// TwinCAT 3 PLC project TcLog_Test
// ProgramVersion: 3.1.4026.20
// libraries:
//   Tc2_Standard, * (Beckhoff Automation GmbH)
//   Tc2_System, * (Beckhoff Automation GmbH)
//   Tc2_Utilities, * (Beckhoff Automation GmbH)
//   Tc3_Module, * (Beckhoff Automation GmbH)
//   [TcLog], * (Benedikt Geisler)
//   TcUnit, * (www.tcunit.org)
// project tree:
//   Tasks/ PlcTask.TcTTO
//   TestRunners/ TestRunner.TcPOU, TestWrapper.TcPOU
//   Tests/ ConvertAnyToString_Test.TcPOU, DateTime_Test.TcPOU, DynamicStringBuffer_Test.TcPOU
// real-time tasks:
//   TASK PlcTask1: cycle T#10ms, priority 21, ADS port 351

CONFIGURATION TcLog_Test
    RESOURCE PLC ON TwinCAT3
        TASK PlcTask(INTERVAL := T#10ms, PRIORITY := 21);
        PROGRAM TestRunner WITH PlcTask : TestRunner;
    END_RESOURCE
END_CONFIGURATION

// ---- TestRunners/TestRunner.TcPOU
PROGRAM TestRunner
VAR
	test_wrapper : TestWrapper;
	date_time_time : DateTime_Test;
	helper_functions_test : ConvertAnyToString_Test;
	dynamic_string_buffer_test : DynamicStringBuffer_Test;
END_VAR

test_wrapper();

TcUnit.Run();

END_PROGRAM

// ---- TestRunners/TestWrapper.TcPOU
FUNCTION_BLOCK TestWrapper
VAR
	core_logger : TcLogCore(BufferSize:=50 * 50 * (Tc2_System.MAX_STRING_LENGTH + Constants.FifoOverhead));
	core_logger_first_cycle : TcLogCore(BufferSize:=50 * 50 * (Tc2_System.MAX_STRING_LENGTH + Constants.FifoOverhead));
	core_logger_first_cycle_valid_timestamp_only : TcLogCore(BufferSize:=50 * 50 * (Tc2_System.MAX_STRING_LENGTH + Constants.FifoOverhead));
	logger_first_cycle : TcLog;
	logger_first_cycle_valid_timestamp_only : TcLog;
	logger : TcLog;
	flush_cache : BOOL;
	ads_adapter : AdsLogTargetAdapter;
 
	// Test drivers
	date_time : DateTime;
	set_local_system_time : NT_SetLocalTime;
	cycles : INT;
	_i : INT;
	persistence_time_stays_within_bounds : F_Trig;
	is_first_cycle: BOOL := TRUE;
	
	// Exchanged variables with .NET tests
	FilePath : STRING;
	FileName : STRING;
	Delimiter : STRING(1);
	NewLocalSystemTimeToBeSet : STRING;
	TriggerNewLocalSystemTime : BOOL;
	LocalTimeAsString : STRING;
	
	Persist_simple_error_message_run : BOOL;
	Persist_simple_error_message_data : STRING;
	
	Persist_long_error_message_run : BOOL;
	Persist_long_error_message_data : T_MaxString;
	
	Linebreak_is_included_when_log_message_has_maximum_length_run : BOOL;
	Linebreak_is_included_when_log_message_has_maximum_length_data : T_MaxString;
	
	Do_not_persist_logs_below_log_level_run : BOOL;
	
	Log_message_contains_instance_path_run : BOOL;
	
	Log_message_uses_correct_delimiter_run : BOOL;
	Log_message_uses_correct_delimiter_data : STRING;
	
	Log_message_contains_custom_formatted_timestamp_run : BOOL;
	
	Delete_logs_if_expired_run : BOOL;
	
	New_logfile_is_created_if_rolling_interval_rolls_run : BOOL;
	
	Same_log_file_is_used_until_rolling_interval_rolls : BOOL;
	
	Log_in_consecutive_cycles : BOOL;
	Number_of_log_cycles : DINT;
	
	Log_multiple_logs_in_one_cycle : BOOL;
	Number_of_logs_per_cycle : DINT;
	
	Log_multiple_logs_in_multiple_cycles : BOOL;
	Number_of_cycles : DINT;
	CycleCount : DINT := 1;
	
	Persistance_time_stays_within_bounds : BOOL;
	Duration_in_cylces : DINT := 1;
END_VAR

// ****** U N I T   T E S T S ******

// Set up TcLog
core_logger
	.IncludeInstancePath()
	.MinimumLevel(LogLevel.Debug)
	.SetDelimiter(Delimiter)
	.SetRollingInterval(RollingIntervals.Hourly)
	.DeleteLogFilesAfterDays(1)
	.TimestampFormat('_YYMMDD-hh-mm-ss_')
	.WriteToAds()
	.WriteToFile('C:\Log Files', 'tclog_test.log')
	.WriteToAdapter(ads_adapter)
	.RunLogger();
//logger.SetLogger(core_logger);

IF flush_cache THEN
	core_logger.FlushCache();
END_IF
  
// Test drivers
date_time.CyclicCall();
LocalTimeAsString := date_time.AsLocalSystemTimeString;

set_local_system_time(
	NetId   := '',
	TimeStr := STRING_TO_SYSTEMTIME(NewLocalSystemTimeToBeSet),
	Start   := TriggerNewLocalSystemTime,
	TmOut := T#2S
);

// Execute tests
IF Persist_simple_error_message_run THEN
	Persist_simple_error_message_run := FALSE;
	logger.Error(Persist_simple_error_message_data);
END_IF

IF Persist_long_error_message_run THEN
	Persist_long_error_message_run := FALSE;
	logger.ToCustomFormat(Persist_long_error_message_data);
END_IF

IF Linebreak_is_included_when_log_message_has_maximum_length_run THEN
	Linebreak_is_included_when_log_message_has_maximum_length_run := FALSE;
	logger
		.ToCustomFormat(Linebreak_is_included_when_log_message_has_maximum_length_data);
	logger.ToCustomFormat(Linebreak_is_included_when_log_message_has_maximum_length_data);
END_IF

IF Do_not_persist_logs_below_log_level_run THEN
	Do_not_persist_logs_below_log_level_run := FALSE;
	logger.Information('Nothing');
END_IF

IF Log_message_contains_instance_path_run THEN
	Log_message_contains_instance_path_run := FALSE;
	logger.Error('Nothing');
END_IF

IF Log_message_uses_correct_delimiter_run THEN
	Log_message_uses_correct_delimiter_run := FALSE;
	logger.Error(Log_message_uses_correct_delimiter_data);
END_IF

IF Log_message_contains_custom_formatted_timestamp_run THEN
	Log_message_contains_custom_formatted_timestamp_run := FALSE;
	logger.Error('Test message');
END_IF

IF Delete_logs_if_expired_run THEN
	Delete_logs_if_expired_run := FALSE;
	logger.Error('Test message');
END_IF

IF New_logfile_is_created_if_rolling_interval_rolls_run THEN
	New_logfile_is_created_if_rolling_interval_rolls_run := FALSE;
	logger.Error('Test message');
END_IF

IF Same_log_file_is_used_until_rolling_interval_rolls THEN
	Same_log_file_is_used_until_rolling_interval_rolls := FALSE;
	logger.Error('Test message');
END_IF

IF Log_in_consecutive_cycles THEN
	logger.Error(Tc2_Standard.CONCAT('Logging cycle ', INT_TO_STRING(cycles)));
	cycles := cycles + 1;
	IF cycles >= Number_of_log_cycles THEN
		cycles := 0;
		Log_in_consecutive_cycles := FALSE;
	END_IF
END_IF

IF Log_multiple_logs_in_one_cycle THEN
	FOR _i:= 1 TO DINT_TO_INT(Number_of_logs_per_cycle) DO
		logger.
			Error(Tc2_Standard.CONCAT('Logging multiple times per cycle. Current step: ', INT_TO_STRING(_i))); 
	END_FOR
	Log_multiple_logs_in_one_cycle := FALSE;
END_IF

IF Log_multiple_logs_in_multiple_cycles THEN
	IF CycleCount <= Number_of_cycles THEN  
		FOR _i:= 1 TO DINT_TO_INT(Number_of_logs_per_cycle) DO
			logger
				.AppendString('Logging multiple times per cycle. Cycle: ')
				.AppendString(DINT_TO_STRING(CycleCount))
				.AppendString(' / Step: ')
				.AppendString(INT_TO_STRING(_i))
				.Error('');
		END_FOR
		CycleCount := CycleCount + 1;
	ELSE
		CycleCount := 1;
		Log_multiple_logs_in_multiple_cycles := FALSE;
	END_IF
END_IF 

persistence_time_stays_within_bounds(CLK := (Persistance_time_stays_within_bounds AND core_logger.Busy));
IF persistence_time_stays_within_bounds.Q THEN
	CycleCount := 1;
	Persistance_time_stays_within_bounds := FALSE;
END_IF

IF Persistance_time_stays_within_bounds THEN
	Duration_in_cylces := Duration_in_cylces + 1;
	IF CycleCount <= Number_of_cycles THEN  
		FOR _i:= 1 TO DINT_TO_INT(Number_of_logs_per_cycle) DO
			logger
				.AppendString('Logging multiple times per cycle. Cycle: ')
				.AppendString(DINT_TO_STRING(CycleCount))
				.AppendString(' / Step: ')
				.AppendString(INT_TO_STRING(_i))
				.Error('');
		END_FOR
		CycleCount := CycleCount + 1;
	END_IF
END_IF

// Check first cpu cycle
core_logger_first_cycle
	.IncludeInstancePath()
	.MinimumLevel(LogLevel.Warning)
	.SetDelimiter(Delimiter)
	.SetRollingInterval(RollingIntervals.Hourly)
	.DeleteLogFilesAfterDays(1)
	.TimestampFormat('_YYYYMMDD-hh-mm-ss_')
	.WriteToAds()
	.WriteToFile('C:\UnitTestFirstCycle\', 'firstCycle.txt')
	.RunLogger();
logger_first_cycle.SetLogger(core_logger_first_cycle);

core_logger_first_cycle_valid_timestamp_only
	.IncludeInstancePath()
	.MinimumLevel(LogLevel.Warning)
	.SetDelimiter(Delimiter)
	.SetRollingInterval(RollingIntervals.Hourly)
	.DeleteLogFilesAfterDays(1)
	.TimestampFormat('_YYYYMMDD-hh-mm-ss_')
	.WriteToAds()
	.WriteToFile('C:\UnitTestFirstCycle\', 'firstCycleValidTimestampOnly.txt')
	.ValidTimestampsOnly()
	.RunLogger();
logger_first_cycle_valid_timestamp_only.SetLogger(core_logger_first_cycle_valid_timestamp_only);

IF is_first_cycle THEN
	logger_first_cycle.Error('Log in first cycle');
	logger_first_cycle_valid_timestamp_only.Error('Log in first cycle with valid timestamps only');
	is_first_cycle := FALSE;
END_IF

END_FUNCTION_BLOCK

// ---- Tests/DateTime_Test.TcPOU
FUNCTION_BLOCK DateTime_Test EXTENDS TcUnit.FB_TestSuite

CheckStringFormat();

METHOD CheckStringFormat
VAR_INST
	date_time : DateTime;
	expected : STRING;
	result : STRING;
END_VAR
VAR
	local_system_time : Tc2_Utilities.TimeStruct;
END_VAR
date_time.CyclicCall();

Test('CheckStringFormat');

local_system_time := date_time.AsLocalSystemTime;

expected := Tc2_Standard.CONCAT('-', TO_STRING(local_system_time.wYear));
IF local_system_time.wMonth < 10 THEN
	expected := Tc2_Standard.CONCAT(expected, '0');
END_IF

expected := Tc2_Standard.CONCAT(expected, TO_STRING(local_system_time.wMonth));
IF local_system_time.wDay < 10 THEN
	expected := Tc2_Standard.CONCAT(expected, '0');
END_IF

expected := Tc2_Standard.CONCAT(expected, TO_STRING(local_system_time.wDay));
expected := Tc2_Standard.CONCAT(expected, '-');
IF local_system_time.wHour < 10 THEN
	expected := Tc2_Standard.CONCAT(expected, '0');
END_IF

expected := Tc2_Standard.CONCAT(expected, TO_STRING(local_system_time.wHour));
expected := Tc2_Standard.CONCAT(expected, ':');
IF local_system_time.wMinute < 10 THEN 
	expected := Tc2_Standard.CONCAT(expected, '0');
END_IF

expected := Tc2_Standard.CONCAT(expected, TO_STRING(local_system_time.wMinute));
expected := Tc2_Standard.CONCAT(expected, ':');
IF local_system_time.wSecond < 10 THEN
	expected := Tc2_Standard.CONCAT(expected, '0');
END_IF

expected := Tc2_Standard.CONCAT(expected, TO_STRING(local_system_time.wSecond));
expected := Tc2_Standard.CONCAT(expected, '-');
result := date_time.ToFormatString('-YYYYMMDD-hh:mm:ss-');
IF date_time.Done THEN
	AssertEquals(
		Expected  :=  expected,
		Actual    :=  result,
		Message   :=  'Time formatting failed.'
	);

  Test_Finished();
END_IF
END_METHOD

END_FUNCTION_BLOCK

// ---- Tests/ConvertAnyToString_Test.TcPOU
FUNCTION_BLOCK ConvertAnyToString_Test EXTENDS TcUnit.FB_TestSuite

ConvertAnyByteToString();
ConvertAnyDateAndTimeToString();
ConvertAnyDateToString();
ConvertAnyDIntToString();
ConvertAnyDTToString();
ConvertAnyIntToString();
ConvertAnyLIntToString();
//ConvertAnyLRealToString();
ConvertAnyLWordToString();
ConvertAnyRealToString();
ConvertAnySIntToString();
ConvertAnyStringToString();
ConvertAnyTimeToString();
ConvertAnyTODToString();
ConvertAnyUDIntToString();
ConvertAnyUIntToString();
ConvertAnyULIntToString();
ConvertAnyUSIntToString();
ConvertAnyWordToString();
ConvertAnyWStringToString();

METHOD ConvertAnyByteToString : BOOL
VAR
	inputs : ARRAY[1..4] OF BYTE := [0, 1, 128, 255];
	expectedValues : ARRAY[1..4] OF STRING := ['0', '1', '128', '255'];
	results : ARRAY[1..4] OF STRING;
	i: INT;
END_VAR
TEST('ConvertAnyByteToString');
 
FOR i := 1 TO 4 DO
  results[i] := AnyToString(inputs[i]);
  AssertEquals(Expected := expectedValues[i],
             Actual := results[i],
             Message := FormatResult(expectedValues[i], results[i])); 
END_FOR
 
TEST_FINISHED();
END_METHOD

METHOD ConvertAnyDateAndTimeToString : BOOL
VAR
	input : DATE_AND_TIME := DT#1970-01-01-00:00;
	result : STRING;
	expected : STRING := 'DT#1970-01-01-00:00:00';
END_VAR
TEST('ConvertAnyDateAndTimeToString');
 
result := AnyToString(input);
 
AssertEquals(Expected := expected,
             Actual := result,
             Message := FormatResult(expected, result));
 
TEST_FINISHED();
END_METHOD

METHOD ConvertAnyDateToString : BOOL
VAR
	input : DATE := D#1970-01-01;
	result : STRING;
	expected : STRING := 'D#1970-01-01';
END_VAR
TEST('ConvertAnyDateToString');
 
result := AnyToString(input);
 
AssertEquals(Expected := expected,
             Actual := result,
             Message := FormatResult(expected, result));
 
TEST_FINISHED();
END_METHOD

METHOD ConvertAnyDIntToString : BOOL
VAR
	inputs : ARRAY[1..7] OF DINT := [-2147483648, -1073741824, -1, 0, 1, 1073741824, 2147483647];
	expectedValues : ARRAY[1..7] OF STRING := ['-2147483648', '-1073741824', '-1', '0', '1', '1073741824', '2147483647'];
	results : ARRAY[1..7] OF STRING;
	i: INT;
END_VAR
TEST('ConvertAnyDINTToString');
 
FOR i := 1 TO 7 DO
  results[i] := AnyToString(inputs[i]);
  AssertEquals(Expected := expectedValues[i],
             Actual := results[i],
             Message := FormatResult(expectedValues[i], results[i])); 
END_FOR

TEST_FINISHED();
END_METHOD

METHOD ConvertAnyDTToString : BOOL
VAR
	input : DT := DT#1970-01-01-00:00;
	result : STRING;
	expected : STRING := 'DT#1970-01-01-00:00:00';
END_VAR
TEST('ConvertAnyDateTimeToString');
 
result := AnyToString(input);
 
AssertEquals(Expected := expected,
             Actual := result,
             Message := FormatResult(expected, result));
 
TEST_FINISHED();
END_METHOD

METHOD ConvertAnyDWordToString : BOOL
VAR
	inputs : ARRAY[1..4] OF DWORD := [0, 1, 2147483647, 4294967295];
	expectedValues : ARRAY[1..4] OF STRING := ['0', '1', '2147483647', '4294967295'];
	results : ARRAY[1..4] OF STRING;
	i: INT;
END_VAR
TEST('ConvertAnyDWordToString');
 
FOR i := 1 TO 4 DO
  results[i] := AnyToString(inputs[i]);
  AssertEquals(Expected := expectedValues[i],
             Actual := results[i],
             Message := FormatResult(expectedValues[i], results[i])); 
END_FOR
 
TEST_FINISHED();
END_METHOD

METHOD ConvertAnyIntToString : BOOL
VAR
	inputs : ARRAY[1..7] OF INT := [-32768, -18000, -1, 0, 1, 18000, 32767];
	expectedValues : ARRAY[1..7] OF STRING := ['-32768', '-18000', '-1', '0', '1', '18000', '32767'];
	results : ARRAY[1..7] OF STRING;
	i: INT;
END_VAR
TEST('ConvertAnyINTToString');

FOR i := 1 TO 7 DO
  results[i] := AnyToString(inputs[i]);
  AssertEquals(Expected := expectedValues[i],
             Actual := results[i],
             Message := FormatResult(expectedValues[i], results[i])); 
END_FOR
      
TEST_FINISHED();
END_METHOD

METHOD ConvertAnyLIntToString : BOOL
VAR
	inputs : ARRAY[1..7] OF LINT := [-2147483648, -18000, -1, 0, 1, 18000, 2147483648];
	expectedValues : ARRAY[1..7] OF STRING := ['-2147483648', '-18000', '-1', '0', '1', '18000', '2147483648'];
	results : ARRAY[1..7] OF STRING;
	i: INT;
END_VAR
TEST('ConvertAnyLINTToString');
 
FOR i := 1 TO 7 DO
  results[i] := AnyToString(inputs[i]);
  AssertEquals(Expected := expectedValues[i],
             Actual := results[i],
             Message := FormatResult(expectedValues[i], results[i])); 
END_FOR
 
TEST_FINISHED();
END_METHOD

METHOD ConvertAnyLRealToString : BOOL
VAR
	inputs : ARRAY[1..5] OF LREAL := [-1.7976931348623157E+308, -4.94065645841247E-324, 0, 4.94065645841247E-324, 1.7976931348623157E+308];
	expectedValues : ARRAY[1..5] OF STRING := ['-1.7976931348623157E308', '-4.94065645841247E324', '0.0', '4.94065645841247E324', '1.7976931348623157E308'];
	results : ARRAY[1..5] OF STRING;
	i: INT;
END_VAR
TEST('ConvertAnyRealToString');
 
FOR i := 1 TO 5 DO
  results[i] := AnyToString(inputs[i]);
  AssertEquals(Expected := expectedValues[i],
             Actual := results[i],
             Message := FormatResult(expectedValues[i], results[i])); 
END_FOR
 
TEST_FINISHED();
END_METHOD

METHOD ConvertAnyLWordToString : BOOL
VAR
	inputs : ARRAY[1..4] OF LWORD := [0, 1, 2147483647, 4294967295];
	expectedValues : ARRAY[1..4] OF STRING := ['0', '1', '2147483647', '4294967295'];
	results : ARRAY[1..4] OF STRING;
	i: INT;
END_VAR
TEST('ConvertAnyLWordToString');
 
FOR i := 1 TO 4 DO
  results[i] := AnyToString(inputs[i]);
  AssertEquals(Expected := expectedValues[i],
             Actual := results[i],
             Message := FormatResult(expectedValues[i], results[i])); 
END_FOR

TEST_FINISHED();
END_METHOD

METHOD ConvertAnyRealToString : BOOL
VAR
	inputs : ARRAY[1..5] OF REAL := [-3.402823E+38, -1.0, 0, 1.0, 3.402823E+38];
	expectedValues : ARRAY[1..5] OF STRING := ['-3.402823E38', '-1.0', '0.0', '1.0', '3.402823E38'];
	results : ARRAY[1..5] OF STRING;
	i: INT;
END_VAR
TEST('ConvertAnyRealToString');
 
FOR i := 1 TO 5 DO
  results[i] := AnyToString(inputs[i]);
  AssertEquals(Expected := expectedValues[i],
             Actual := results[i],
             Message := FormatResult(expectedValues[i], results[i])); 
END_FOR
 
TEST_FINISHED();
END_METHOD

METHOD ConvertAnySIntToString : BOOL
VAR
	inputs : ARRAY[1..5] OF SINT := [-128, -1, 0, 1, 127];
	expectedValues : ARRAY[1..5] OF STRING := ['-128', '-1', '0', '1', '127'];
	results : ARRAY[1..5] OF STRING;
	i: INT;
END_VAR
TEST('ConvertAnySINTToString');
 
FOR i := 1 TO 5 DO
  results[i] := AnyToString(inputs[i]);
  AssertEquals(Expected := expectedValues[i],
             Actual := results[i],
             Message := FormatResult(expectedValues[i], results[i])); 
END_FOR
 
TEST_FINISHED();
END_METHOD

METHOD ConvertAnyStringToString : BOOL
VAR
	input : STRING := 'Hallo';
	result : STRING;
	expected : STRING := 'Hallo';
END_VAR
TEST('ConvertAnyStringToString');
 
result := AnyToString(input);
 
AssertEquals(Expected := expected,
             Actual := result,
             Message := FormatResult(expected, result));
 
TEST_FINISHED();
END_METHOD

METHOD ConvertAnyTimeToString : BOOL
VAR
	input : TIME := T#49D17H2M47S295MS;
	result : STRING;
	expected : STRING := 'T#49d17h2m47s295ms';
END_VAR
TEST('ConvertAnyTimeToString');
 
result := AnyToString(input);
 
AssertEquals(Expected := expected,
             Actual := result,
             Message := FormatResult(expected, result));
 
TEST_FINISHED();
END_METHOD

METHOD ConvertAnyTODToString : BOOL
VAR
	input : TOD := TOD#11:02:47.295;
	result : STRING;
	expected : STRING := 'TOD#11:02:47.295';
END_VAR
TEST('ConvertAnyTODToString');
 
result := AnyToString(input);
 
AssertEquals(Expected := expected,
             Actual := result,
             Message := FormatResult(expected, result));
 
TEST_FINISHED();
END_METHOD

METHOD ConvertAnyUDIntToString : BOOL
VAR
	inputs : ARRAY[1..3] OF UDINT := [0, 1, 4294967295];
	expectedValues : ARRAY[1..3] OF STRING := ['0', '1', '4294967295'];
	results : ARRAY[1..3] OF STRING;
	i: INT;
END_VAR
TEST('ConvertAnyUDINTToString');

FOR i := 1 TO 3 DO
  results[i] := AnyToString(inputs[i]);
  AssertEquals(Expected := expectedValues[i],
             Actual := results[i],
             Message := FormatResult(expectedValues[i], results[i])); 
END_FOR
 
TEST_FINISHED();
END_METHOD

METHOD ConvertAnyUIntToString : BOOL
VAR
	inputs : ARRAY[1..3] OF UINT := [0, 1, 65535];
	expectedValues : ARRAY[1..3] OF STRING := ['0', '1', '65535'];
	results : ARRAY[1..3] OF STRING;
	i: INT;
END_VAR
TEST('ConvertAnyUINTToString');
 
FOR i := 1 TO 3 DO
  results[i] := AnyToString(inputs[i]);
  AssertEquals(Expected := expectedValues[i],
             Actual := results[i],
             Message := FormatResult(expectedValues[i], results[i])); 
END_FOR
 
TEST_FINISHED();
END_METHOD

METHOD ConvertAnyULIntToString : BOOL
VAR
	inputs : ARRAY[1..3] OF ULINT := [0, 1, 4294967295];
	expectedValues : ARRAY[1..3] OF STRING := ['0', '1', '4294967295'];
	results : ARRAY[1..3] OF STRING;
	i: INT;
END_VAR
TEST('ConvertAnyULINTToString');
 
FOR i := 1 TO 3 DO
  results[i] := AnyToString(inputs[i]);
  AssertEquals(Expected := expectedValues[i],
             Actual := results[i],
             Message := FormatResult(expectedValues[i], results[i])); 
END_FOR
 
TEST_FINISHED();
END_METHOD

METHOD ConvertAnyUSIntToString : BOOL
VAR
	inputs : ARRAY[1..3] OF USINT := [0, 1, 255];
	expectedValues : ARRAY[1..3] OF STRING := ['0', '1', '255'];
	results : ARRAY[1..3] OF STRING;
	i: INT;
END_VAR
TEST('ConvertAnyUSINTToString');
 
FOR i := 1 TO 3 DO
  results[i] := AnyToString(inputs[i]);
  AssertEquals(Expected := expectedValues[i],
             Actual := results[i],
             Message := FormatResult(expectedValues[i], results[i])); 
END_FOR
 
TEST_FINISHED();
END_METHOD

METHOD ConvertAnyWordToString : BOOL
VAR
	inputs : ARRAY[1..3] OF WORD := [0, 1, 65535];
	expectedValues : ARRAY[1..3] OF STRING := ['0', '1', '65535'];
	results : ARRAY[1..3] OF STRING;
	i: INT;
END_VAR
TEST('ConvertAnyWordToString');
 
FOR i := 1 TO 3 DO
  results[i] := AnyToString(inputs[i]);
  AssertEquals(Expected := expectedValues[i],
             Actual := results[i],
             Message := FormatResult(expectedValues[i], results[i])); 
END_FOR
 
TEST_FINISHED();
END_METHOD

METHOD ConvertAnyWStringToString : BOOL
VAR
	input : WSTRING := "Hallo";
	result : STRING;
	expected : STRING := 'Hallo';
END_VAR
TEST('ConvertAnyWStringToString');
 
result := AnyToString(input);
 
AssertEquals(Expected := expected,
             Actual := result,
             Message := FormatResult(expected, result));
 
TEST_FINISHED();
END_METHOD

METHOD PRIVATE FormatResult : STRING
VAR_INPUT
	Expected : STRING;
	Result : STRING;
END_VAR
FormatResult := Tc2_Standard.CONCAT('Conversion failed. Expected: ', Tc2_Standard.CONCAT(Expected, Tc2_Standard.CONCAT(' - Result: ', Result)));
END_METHOD

END_FUNCTION_BLOCK

// ---- Tests/DynamicStringBuffer_Test.TcPOU
FUNCTION_BLOCK DynamicStringBuffer_Test EXTENDS FB_TestSuite

LogsManyMessagesForManyCycles();

METHOD LogsManyMessagesForManyCycles
VAR
	result : STRING := '';
	expected : STRING := '';
	i : UDINT;
END_VAR
VAR CONSTANT
	Cycles : UDINT := 50;
	Messages : UDINT := 50;
END_VAR
VAR_INST
	cycleCount : UDINT := 0;
	logsManyMessagesForManyCyclesLogger : TcLogCore(BufferSize:=50 * 50 * 280); // Cycles * Messages * (max string length + fifo overhead (estimated))
	logger : TcLog;
END_VAR
Test('LogsManyMessagesForManyCycles');

logsManyMessagesForManyCyclesLogger
  .WriteToFile('c:\UnitTest\', 'test.txt')
  .RunLogger();
logger.SetLogger(logsManyMessagesForManyCyclesLogger);

IF cycleCount < Cycles THEN
  FOR i:=0 TO Messages DO
    logger
      .AppendString('Cycle: ')
      .AppendString(UDINT_TO_STRING(cycleCount))
      .AppendString(', Message: ')
      .AppendString(UDINT_TO_STRING(i))
      .Error(''); 
  END_FOR
END_IF
cycleCount := cycleCount + 1;

// Catch any occuring error message
IF LEN(logsManyMessagesForManyCyclesLogger.Error.Info) > 0 THEN
  result := logsManyMessagesForManyCyclesLogger.Error.Info;
END_IF

IF cycleCount > (Cycles * Messages * 2 + 4) THEN 
  AssertEquals(Expected := expected,
         Actual := result,
         Message := result);
 
  Test_Finished();
END_IF
END_METHOD

END_FUNCTION_BLOCK
